FUNCTION IsOk : BOOL
VAR_INPUT
	nIn				: Result;
END_VAR
VAR_OUTPUT
	nOut			: Result;
END_VAR

IsOk := nIn > 0;
nOut := nIn;

END_FUNCTION

(* stored: Version 1.1.0.1
   POU IsOk: Id {a86826be-b52a-46f1-b35e-fa89d49ee7eb}, SpecialFunc None *)
